PROGRAM dbg_highest
VAR
END_VAR

IF NOT framework_is_local_simulated()
THEN
	RETURN;	
END_IF
dbg_root();
dbg_quality_checks();
dbg_csp_case_closing_ls_horizontal();
dbg_csp_case_closing_ls_lower();
dbg_csp_case_closing_ls_upper();
dbg_csp_case_closing_os_horizontal();
dbg_csp_case_closing_os_lower();
dbg_csp_case_closing_os_upper();
dbg_csp_case_discharge_accu_depth();
dbg_csp_case_discharge_belts_conveyor();
dbg_csp_case_discharge_belts_rotate();
dbg_csp_case_discharge_reject_belt();
dbg_csp_case_discharge_reject_sensors();
dbg_csp_case_discharge_speedbelt_ls();
dbg_csp_case_discharge_speedbelt_os();
dbg_csp_case_feed_arm_elbow();
dbg_csp_case_feed_arm_sensors();
dbg_csp_case_feed_arm_shoulder();
dbg_csp_case_feed_arm_wrist();
dbg_csp_case_feed_kinematic_tilt();
dbg_csp_case_feed_kinematic_x();
dbg_csp_case_feed_kinematic_y();
dbg_csp_case_feed_magazine_accu_lsdepth();
dbg_csp_case_feed_magazine_accu_osdepth();
dbg_csp_case_feed_magazine_level_zone1();
dbg_csp_case_feed_magazine_level_zone2();
dbg_csp_case_feed_magazine_level_zone3();
dbg_csp_case_feed_magazine_level_zonelow();
dbg_csp_case_feed_magazine_level_zonemin();
dbg_csp_case_feed_magazine_ls_belt();
dbg_csp_case_feed_magazine_ls_pusher();
dbg_csp_case_feed_magazine_ls_pushertilt();
dbg_csp_case_feed_magazine_ls_sensors();
dbg_csp_case_feed_magazine_os_belt();
dbg_csp_case_feed_magazine_os_pusher();
dbg_csp_case_feed_magazine_os_pushertilt();
dbg_csp_case_feed_magazine_os_sensors();
dbg_csp_case_feed_reject_belt_lower();
dbg_csp_case_feed_reject_belt_upper();
dbg_csp_case_feed_reject_sensors();
dbg_csp_case_feed_shuttle_accu_depth();
dbg_csp_case_feed_shuttle_horizontal();
dbg_csp_case_feed_shuttle_sensors();
dbg_csp_case_feed_shuttle_sensors_ls();
dbg_csp_case_feed_shuttle_sensors_os();
dbg_csp_case_feed_shuttle_vertical();
dbg_csp_case_fc_ls_lower_follower();
dbg_csp_case_fc_ls_lower_sensors();
dbg_csp_case_fc_ls_lower_spreader();
dbg_csp_case_fc_ls_lower_trailingcloser();
dbg_csp_case_fc_ls_upper_follower();
dbg_csp_case_fc_ls_upper_leadingminorcloser();
dbg_csp_case_fc_ls_upper_sensors();
dbg_csp_case_fc_ls_upper_spreader();
dbg_csp_case_fc_os_lower_follower();
dbg_csp_case_fc_os_lower_sensors();
dbg_csp_case_fc_os_lower_spreader();
dbg_csp_case_fc_os_lower_trailingcloser();
dbg_csp_case_fc_os_upper_follower();
dbg_csp_case_fc_os_upper_sensors();
dbg_csp_case_fc_os_upper_spreader();
dbg_csp_case_glue_hotmelt();
dbg_csp_case_glue_ls_accu_lowerposition();
dbg_csp_case_glue_ls_accu_upperposition();
dbg_csp_case_glue_os_accu_lowerposition();
dbg_csp_case_glue_os_accu_upperposition();
dbg_csp_case_glue_os_accu_width();
dbg_csp_case_glue_virtualmaster();
dbg_csp_case_loader_guide_accu_width();
dbg_csp_case_loader_guide_downstream();
dbg_csp_case_loader_guide_length();
dbg_csp_case_loader_guide_upstream();
dbg_csp_case_main_safety_accuchange();
dbg_csp_case_main_safety_drives_commonconfiguration();
dbg_csp_case_main_safety_drives_ps2000();
dbg_csp_case_main_safety_drives_sd10000();
dbg_csp_case_main_safety_drives_sd10100();
dbg_csp_case_main_safety_drives_sd10200();
dbg_csp_case_main_safety_drives_sd10300();
dbg_csp_case_main_safety_drives_sd10400();
dbg_csp_case_main_safety_drives_sd11000();
dbg_csp_case_main_safety_drives_sd12000();
dbg_csp_case_main_safety_drives_sd15000();
dbg_csp_case_main_safety_drives_sd2100();
dbg_csp_case_main_safety_drives_sd2200();
dbg_csp_case_main_safety_drives_sd2300();
dbg_csp_case_main_safety_drives_sd2400();
dbg_csp_case_main_safety_drives_sd2500();
dbg_csp_case_main_safety_drives_sd26000();
dbg_csp_case_main_safety_drives_sd26100();
dbg_csp_case_main_safety_drives_sd8000();
dbg_csp_case_main_safety_drives_sd8100();
dbg_csp_case_main_safety_drives_sd8200();
dbg_csp_case_main_safety_drives_sd8300();
dbg_csp_case_main_safety_drives_sd8400();
dbg_csp_case_main_safety_drives_sd8500();
dbg_csp_case_main_safety_drives_sd8600();
dbg_csp_case_main_safety_emergency();
dbg_csp_case_main_safety_guards();
dbg_csp_case_openflap_sensors();
dbg_csp_case_tr_accu_depth();
dbg_csp_case_tr_accu_ls_width();
dbg_csp_case_tr_accu_os_width();
dbg_csp_case_tr_squaring_ls_leading();
dbg_csp_case_tr_squaring_ls_trailing();
dbg_csp_case_tr_squaring_os_leading();
dbg_csp_case_tr_squaring_os_trailing();
dbg_csp_case_transport_accu_depth();
dbg_csp_case_transport_ls_leading();
dbg_csp_case_transport_ls_trailing();
dbg_csp_case_transport_os_leading();
dbg_csp_case_transport_os_minorplow();
dbg_csp_case_transport_os_trailing();
dbg_csp_case_transport_virtualmaster();
dbg_csp_main_motorization_virtualmanager();
dbg_csp_transfer_accumulator_accu_convdepth();
dbg_csp_transfer_accumulator_accu_depth();
dbg_csp_transfer_accumulator_accu_topraillength();
dbg_csp_transfer_accumulator_accu_toprailwidth();
dbg_csp_transfer_accumulator_belt();
dbg_csp_transfer_accumulator_finger_ls();
dbg_csp_transfer_accumulator_finger_os();
dbg_csp_transfer_accumulator_lift();
dbg_csp_transfer_accumulator_virtualmaster();
dbg_csp_transfer_infeed();

END_PROGRAM

(* stored: Version 1.1.0.1, ProductVersion 3.1.4022.12
   POU dbg_highest: Id {73cb7746-8b0d-4bb2-bd41-8cad5e1554cf}, SpecialFunc None *)
